(* LS Electric XG5000 project: PID TEST *)
(* PLC NewPLC *)
(* module base 0 slot 0: 입출력 모듈:XEM-DN/DP32H2 (DC 24V 입력, 트랜지스터 출력 32점 (싱크출력/소스출력)) *)
(* module base 0 slot 1: 내장위치결정:XBF-PO02E (오픈컬렉터형, 2축) *)
(* module base 0 slot 2: Cnet:XBL-C41A (Cnet 통신 모듈(RS-422/485)) *)
(* module base 0 slot 3: Cnet:XBL-C41A (Cnet 통신 모듈(RS-422/485)) *)

FUNCTION FC_SCP : REAL
VAR_INPUT
    X : REAL;
    X_MX : REAL;
    X_MN : REAL;
    Y_MX : REAL;
    Y_MN : REAL;
END_VAR
VAR
    Y : REAL;
END_VAR
Y := ((X - X_MN) * ((Y_MX - Y_MN) / (X_MX - X_MN))) + Y_MN;
FC_SCP:= Y;
END_FUNCTION

FUNCTION_BLOCK FB_MDOL
(* Motor Control D.O.L *)
VAR_INPUT
    I_REM : BOOL; (* Remote Select (PLC) *)
    A_SEL : BOOL; (* Auto Select (HMI) *)
    M_SEL : BOOL; (* Manual Select (HMI) *)
    A_STT : BOOL; (* Start Command (Logic) *)
    M_STT : BOOL; (* Start Command (HMI) *)
    M_STP : BOOL; (* Stop Command (HMI) *)
    I_TPS : BOOL; (* Test Position (PLC) *)
    I_RUN : BOOL; (* Run Feedback (PLC) *)
    I_FLT : BOOL; (* Fault (PLC) *)
END_VAR
VAR_OUTPUT
    REM : BOOL; (* Remote Mode (HMI) *)
    AT : BOOL; (* Auto Mode (HMI) *)
    TPOS : BOOL; (* Test Positon (HMI) *)
    PMSV : BOOL; (* Start Permissive (HMI) *)
    Q_RUN : BOOL; (* Start - Latch (PLC) *)
    Q_STT : BOOL; (* Start - Pulse (PLC) *)
    Q_STP : BOOL; (* Stop - Pulse (PLC) *)
    RUN : BOOL; (* Run (HMI) *)
    FLT : BOOL; (* Fault (HMI) *)
    ALM : BOOL; (* Alarm (HMI) *)
END_VAR
VAR
    TON_ALM : TON;
    TP_STP : TP;
    TP_STT : TP;
END_VAR
// 2021.08.10 PKD
// FUNCTION BLOCK - MOTOR (DOL)

REM:= I_REM;
PMSV:= NOT(FLT) AND NOT(I_FLT) AND NOT(Q_RUN);
IF A_SEL THEN
	AT:= TRUE;
ELSIF M_SEL THEN
	AT:= FALSE;
END_IF;


IF (NOT(I_TPS) AND ((REM AND ((NOT(AT) AND M_STT) OR (AT AND A_STT))) OR (NOT(REM) AND I_RUN))) OR (I_TPS AND REM AND M_STT) THEN
	Q_RUN:= TRUE;
ELSIF (NOT(I_TPS) AND ((REM AND ((NOT(AT) AND M_STP) OR (AT AND NOT(A_STT)))) OR (NOT(REM) AND NOT(I_RUN)))) OR (I_TPS AND REM AND M_STP) OR I_FLT THEN
	Q_RUN:= FALSE;
END_IF;

TP_STT(IN:=Q_RUN, PT:=T#3S);
Q_STT:= TP_STT.Q;

TP_STP(IN:=NOT(Q_RUN), PT:=T#3S);
Q_STP:= NOT(TP_STP.Q);

Ton_ALM(IN:=(Q_RUN AND NOT(I_RUN)) OR (NOT(Q_RUN) AND I_RUN), PT:=T#1S);
RUN:= I_RUN;
FLT:= I_FLT;
TPOS:= I_TPS;
ALM:= Ton_ALM.Q;
END_FUNCTION_BLOCK

FUNCTION_BLOCK FB_MPID
(* Motor Control - PID *)
VAR_INPUT
    I_REM : BOOL;
    A_SEL : BOOL;
    M_SEL : BOOL;
    A_STT : BOOL; (* AUTO START CMD *)
    M_STT : BOOL; (* MANUAL START CMD *)
    M_STP : BOOL; (* MANUAL STOP CMD *)
    I_TPS : BOOL; (* MCC TEST POSITION SIGNAL *)
    I_RUN : BOOL; (* MCC RUN FEEDBACK SIGNAL *)
    I_FLT : BOOL; (* MCC FAULT SIGNAL *)
    BLK : UINT;
    LOOP : UINT;
    PV : REAL;
    SP : REAL;
    KP : REAL;
    TI : REAL;
    TD : REAL;
    TS : REAL;
    MV_MAX : REAL;
    MV_MIN : REAL;
    MV_DLY : REAL;
    MV_MAN_ON : BOOL;
    PID_MV : INT;
    PV_MAX : REAL;
    PV_MIN : REAL;
    REV : BOOL;
END_VAR
VAR_IN_OUT
    MV_MAN : REAL;
END_VAR
VAR_OUTPUT
    REM : BOOL;
    AT : BOOL;
    TPOS : BOOL; (* MCC TEST POSITION *)
    PMSV : BOOL; (* START StartPmsv *)
    Q_RUN : BOOL; (* START COMMAND *)
    Q_STT : BOOL; (* START COMMAND (3SEC PULSE H) *)
    Q_STP : BOOL; (* STOP COMMAND (3SEC PULSE L) *)
    RUN : BOOL; (* MOTOR RUN *)
    FLT : BOOL; (* MOTOR FAULT *)
    ALM : BOOL; (* MOTOR FEEDBACK ALARM *)
    OUT : REAL;
    PID_PV : INT;
    PID_SP : INT;
    PID_KP : REAL;
    PID_TI : REAL;
    PID_TD : REAL;
    PID_TS : WORD;
    PID_MV_MAX : INT;
    PID_MV_MIN : INT;
    PID_MV_DLY : INT;
    PID_MAN_ON : BOOL;
    PID_MV_MAN : INT;
    PID_BMPL : BOOL;
    PID_REV : BOOL;
END_VAR
VAR
    DONE : BOOL;
    LW_STAT : WORD;
    MTR_DOL : FB_MDOL;
    PID_RUN : PIDRUN;
END_VAR
// 2021.08.10 PKD
// FUNCTION BLOCK - PID CONTROL (MOTOR)

MTR_DOL(
	EN		:= TRUE, 
	I_REM	:= I_REM, 
	A_SEL	:= A_SEL, 
	M_SEL	:= M_SEL, 
	A_STT	:= A_STT, 
	M_STT	:= M_STT, 
	M_STP	:= M_STP, 
	I_TPS	:= I_TPS, 
	I_RUN	:= I_RUN, 
	I_FLT	:= I_FLT, 
	REM		=> REM, 
	AT		=> AT, 
	TPOS	=> TPOS,
	PMSV	=> PMSV, 
	Q_RUN	=> Q_RUN, 
	Q_STT	=> Q_STT,
	Q_STP	=> Q_STP,
	RUN		=> RUN, 
	ALM		=> ALM, 
	FLT		=> FLT);


PID_MAN_ON:= MV_MAN_ON AND NOT(AT);

PID_RUN(
	REQ			:= RUN, 
	BLOCK		:= 0, 
	LOOP		:= 0, 
	DONE		=> DONE,
	PID_STAT	=> LW_STAT);

PID_SP:= LIMIT(MN:=0, IN:=REAL_TO_INT(FC_SCP(X:=SP, X_MX:=PV_MAX, X_MN:=PV_MIN, Y_MX:=4000.0, Y_MN:=0.0)), MX:=4000);
PID_PV:= LIMIT(MN:=0, IN:=REAL_TO_INT(FC_SCP(X:=PV, X_MX:=PV_MAX, X_MN:=PV_MIN, Y_MX:=4000.0, Y_MN:=0.0)), MX:=4000);
PID_KP:= KP;
PID_TI:= TI;
PID_TD:= TD;
PID_TS:= INT_TO_WORD(REAL_TO_INT(TS*10.0));

PID_MV_MAX:= REAL_TO_INT(MV_MAX * 100.0);
PID_MV_MIN:= REAL_TO_INT(MV_MIN * 100.0);
PID_MV_DLY:= REAL_TO_INT(MV_DLY * 000.0);
PID_MV_MAN:= REAL_TO_INT(MV_MAN * 100.0);

PID_BMPL:= TRUE;
PID_REV:= REV;

IF Q_RUN THEN
	OUT:= INT_TO_REAL(PID_MV) * 0.01;
ELSE
	OUT:= 0;
END_IF;

IF NOT(PID_MAN_ON) THEN
	MV_MAN:= OUT;
END_IF;
END_FUNCTION_BLOCK

PROGRAM pidmvtest (* task: 스캔 프로그램 *)
VAR
    CoolAirBlwr_Alm : BOOL;
    CoolAirBlwr_AutoMode : BOOL;
    CoolAirBlwr_AutoSel : BOOL;
    CoolAirBlwr_ManSel : BOOL;
    CoolAirBlwr_MaxMv : REAL;
    CoolAirBlwr_MinMv : REAL;
    CoolAirBlwr_PidKp : REAL := 10;
    CoolAirBlwr_PidManMv : REAL;
    CoolAirBlwr_PidManOnCmd : BOOL;
    CoolAirBlwr_PidOut : REAL;
    CoolAirBlwr_PidSpC : REAL := 10;
    CoolAirBlwr_PidTd : REAL;
    CoolAirBlwr_PidTi : REAL;
    CoolAirBlwr_PidTs : REAL := 100;
    CoolAirBlwr_Pmsv : BOOL;
    CoolAirBlwr_RemMode : BOOL;
    CoolAirBlwr_Run : BOOL;
    CoolAirBlwr_StartCmdAuto : BOOL;
    CoolAirBlwr_StartCmdMan : BOOL;
    CoolAirBlwr_StopCmdMan : BOOL;
    dne : BOOL;
    ExhTemp_Pv : REAL := 20;
    INST_FB_MPID : FB_MPID;
    INST_PIDRUN : PIDRUN;
    INST_PIDRUN1 : PIDRUN;
    kkj : INT;
    LW_STAT : WORD;
    MPID_CoolAirBlwr : FB_MPID;
    PID_RUN : PIDRUN;
    run : BOOL;
    StackAirBlwr_Alm : BOOL;
    StackAirBlwr_AutoMode : BOOL;
    StackAirBlwr_AutoSel : BOOL;
    StackAirBlwr_ManMv : REAL;
    StackAirBlwr_ManSel : BOOL;
    StackAirBlwr_MvMin : REAL;
    StackAirBlwr_PidKp : REAL;
    StackAirBlwr_PidManOnCmd : BOOL;
    StackAirBlwr_PidOut : REAL;
    StackAirBlwr_PidSpC : REAL;
    StackAirBlwr_PidTd : REAL;
    StackAirBlwr_PidTi : REAL;
    StackAirBlwr_PidTs : REAL;
    StackAirBlwr_Pmsv : BOOL;
    StackAirBlwr_RemMode : BOOL;
    StackAirBlwr_Run : BOOL;
    StackAirBlwr_StartCmdAuto : BOOL;
    StackAirBlwr_StartCmdMan : BOOL;
    StackAirBlwr_StopCmdMan : BOOL;
    StackSplyAirFlow_Pv : REAL;
    stat : WORD;
END_VAR
MPID_CoolAirBlwr(
	EN			:= TRUE, 
	I_REM		:= TRUE, 
	A_SEL		:= CoolAirBlwr_AutoSel, 
	M_SEL		:= CoolAirBlwr_ManSel, 
	A_STT		:= CoolAirBlwr_StartCmdAuto, 
	M_STT		:= CoolAirBlwr_StartCmdMan, 
	M_STP		:= CoolAirBlwr_StopCmdMan, 
	I_TPS		:= FALSE, 
	I_RUN		:= MPID_CoolAirBlwr.Q_RUN, 
	I_FLT		:= FALSE, 
	BLK			:= 0, 
	LOOP		:= 0, 
	PV			:= CoolAirBlwr_PidSpC, 
	SP			:= ExhTemp_Pv, 
	KP			:= CoolAirBlwr_PidKp, 
	TI			:= CoolAirBlwr_PidTi, 
	TD			:= CoolAirBlwr_PidTd, 
	TS			:= CoolAirBlwr_PidTs, 
	PV_MAX		:= 500.0, 
	PV_MIN		:= 0.0, 
	MV_MAX		:= CoolAirBlwr_MaxMv, 
	MV_MIN		:= CoolAirBlwr_MinMv, 
	MV_DLY		:= 10.0,
	MV_MAN		:= CoolAirBlwr_PidManMv, 
	MV_MAN_ON	:= CoolAirBlwr_PidManOnCmd,
	PID_MV		:= _PID00_MV, 
	REV			:= FALSE, 
	REM			=> CoolAirBlwr_RemMode, 
	AT			=> CoolAirBlwr_AutoMode, 
	PMSV		=> CoolAirBlwr_Pmsv, 
	run			=> CoolAirBlwr_Run, 
	FLT			=> CoolAirBlwr_Alm, 
	OUT			=> CoolAirBlwr_PidOut, 
	PID_PV		=> _PID00_PV, 
	PID_SP		=> _PID00_SV, 
	PID_MV_MAX	=> _PID00_MV_max, 
	PID_MV_MIN	=> _PID00_MV_min, 
	PID_MV_DLY	=> _PID00_d_MV_max,
	PID_MAN_ON	=> _PID00_MAN, 
	PID_MV_MAN	=> _PID00_MV_man, 
	PID_BMPL	=> _PID00_MV_BMPL, 
	PID_REV		=> _PID00_REV);
	
	_PID00_K_p:= CoolAirBlwr_PidKp;
	_PID00_T_i:= CoolAirBlwr_PidTi;
	_PID00_T_d:= CoolAirBlwr_PidTd;
	_PID00_T_s:= INT_TO_WORD(REAL_TO_INT(CoolAirBlwr_PidTs));

	IF _T1S THEN
		kkj:=kkj*2;
	END_IF;
END_PROGRAM

PROGRAM test (* task: 스캔 프로그램 *)
VAR
    D : REAL;
    I : REAL;
    INST : PIDRUN;
    MV : INT;
    MVMAX : INT;
    MVMIN : INT;
    P : REAL;
    PV : INT;
    run : BOOL;
    STAT : WORD;
    SV : INT;
    TS : WORD;
END_VAR

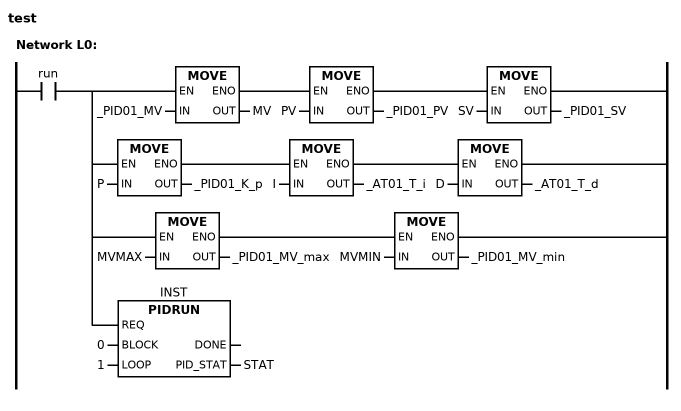
(* Rung L0 *)
IF run THEN
    MV := _PID01_MV;
    _PID01_PV := PV;
    _PID01_SV := SV;
    _PID01_K_p := P;
    _AT01_T_i := I;
    _AT01_T_d := D;
    _PID01_MV_max := MVMAX;
    _PID01_MV_min := MVMIN;
END_IF;
INST(REQ := run, BLOCK := 0, LOOP := 1, PID_STAT => STAT);
END_PROGRAM